Staubli VAL3: ModbusGet.pgx

program modbusGet(num& x_nResult (dimensions=1))
begin
  //start
  if (dStartControl[1]==true and dStartControl[2]==false and dStartControl[3]==false)
    x_nResult=1
    //stop
  elseIf (dStartControl[1]==false and dStartControl[2]==true and dStartControl[3]==false)
    x_nResult=2
    //reset
  elseIf (dStartControl[1]==false and dStartControl[2]==false and dStartControl[3]==true)
    x_nResult=3
    //other
  else
    x_nResult=0
  endIf
end
